// TwinCAT 3 PLC project PlcIotMqttSampleAwsIotShadow
// ProgramVersion: 3.1.4022.7
// libraries:
//   Tc2_Standard, * (Beckhoff Automation GmbH)
//   Tc2_System, * (Beckhoff Automation GmbH)
//   Tc2_Utilities, * (Beckhoff Automation GmbH)
//   Tc3_IotBase, * (Beckhoff Automation GmbH)
//   Tc3_JsonXml, * (Beckhoff Automation GmbH)
//   Tc3_Module, * (Beckhoff Automation GmbH)
// project tree:
//   / PlcTask.TcTTO
//   POUs/ MAIN.TcPOU, PrgMqttCom.TcPOU
// real-time tasks:
//   TASK PlcTask: cycle T#10ms, priority 20, ADS port 350

CONFIGURATION PlcIotMqttSampleAwsIotShadow
    RESOURCE PLC ON TwinCAT3
        TASK PlcTask(INTERVAL := T#10ms, PRIORITY := 20);
        PROGRAM MAIN WITH PlcTask : MAIN;
    END_RESOURCE
END_CONFIGURATION

// ---- POUs/MAIN.TcPOU
PROGRAM MAIN
VAR
	m : INT;
END_VAR

m := m + 1;
PrgMqttCom();

END_PROGRAM

// ---- POUs/PrgMqttCom.TcPOU
PROGRAM PrgMqttCom
VAR
	fbMqttClient 					: FB_IotMqttClient;
	bSetParameter 					: BOOL := TRUE;
	bConnect 						: BOOL := TRUE;
	hrErrorOccurred 				: HRESULT;
	
	(* AWS IoT Shadow  *)
	sTopicShadowUpdate	 			: STRING(255) := '$$aws/things/SvenG-NB05/shadow/update';
	sTopicShadowDocument			: STRING(255) := '$$aws/things/SvenG-NB05/shadow/update/documents';
	sPayloadShadowUpdate			: STRING(1000);
	{attribute 'TcEncoding':='UTF-8'}
	sPayloadShadowDocumentRcv		: STRING(1000);
	bShadowUpdate					: BOOL;
	bShadowDocumentSubscribed		: BOOL;
	
	(* received message and queue handling *)	
	fbMessageQueue 					: FB_IotMqttMessageQueue;
	fbMessage 						: FB_IotMqttMessage;

	(* JSON *)
	fbJson      					: FB_JsonSaxWriter;

END_VAR

IF bSetParameter THEN
	bSetParameter := FALSE;
	
	(* TLS settings for AWS IoT connection *)
	fbMqttClient.stTLS.sCA := 'c:\TwinCAT\3.1\Config\Certificates\AWS\AmazonRootCA1.pem';
    fbMqttClient.stTLS.sCert := 'c:\TwinCAT\3.1\Config\Certificates\AWS\6a1ba937cb-certificate.pem.crt';
    fbMqttClient.stTLS.sKeyFile := 'c:\TwinCAT\3.1\Config\Certificates\AWS\6a1ba937cb-private.pem.key';
	
	(* Broker settings für AWS IoT *)
	fbMqttClient.sHostName:= 'a35rjvy201xp77-ats.iot.eu-central-1.amazonaws.com';
	fbMqttClient.nHostPort:= 8883;
	fbMqttClient.sClientId:= 'SvenG-NB05'; 

	fbMqttClient.ipMessageQueue := fbMessageQueue;
END_IF

fbMqttClient.Execute(bConnect);

IF fbMqttClient.bError THEN
	// add your error logging here
	hrErrorOccurred := fbMqttClient.hrErrorCode;
END_IF
IF fbMessageQueue.nQueuedMessages > 0 THEN
	IF fbMessageQueue.Dequeue(fbMessage:=fbMessage) THEN
		fbMessage.GetTopic(pTopic:=ADR(sTopicShadowDocument), nTopicSize:=SIZEOF(sTopicShadowDocument) );
		fbMessage.GetPayload(pPayload:=ADR(sPayloadShadowDocumentRcv), nPayloadSize:=SIZEOF(sPayloadShadowDocumentRcv), bSetNullTermination:=FALSE);
	END_IF
END_IF

IF fbMqttClient.bConnected THEN
	IF NOT bShadowDocumentSubscribed THEN
		bShadowDocumentSubscribed := fbMqttClient.Subscribe(sTopic:=sTopicShadowDocument, eQoS:=TcIotMqttQos.AtMostOnceDelivery);
		IF fbMqttClient.bError THEN
			// add your error logging here
			hrErrorOccurred := fbMqttClient.hrErrorCode;
		END_IF
	END_IF

	IF bShadowUpdate THEN // update shadow on demand
		bShadowUpdate := FALSE;
		
		// JSON format according to https://docs.aws.amazon.com/iot/latest/developerguide/device-shadow-mqtt.html
		fbJson.StartObject();
		fbJson.AddKey('state');
		fbJson.StartObject();
		fbJson.AddKey('reported');
		fbJson.StartObject();		
		fbJson.AddKey('Vendor');
		fbJson.AddString('Beckhoff Automation');
		fbJson.AddKey('CpuTemperature');
		fbJson.AddDint(42);
		fbJson.AddKey('Operating System');
		fbJson.AddString('FreeBSD');
		fbJson.EndObject();
		fbJson.EndObject();
		fbJson.EndObject();
		sPayloadShadowUpdate := fbJson.GetDocument();
		fbJson.ResetDocument();
	
		fbMqttClient.Publish(	sTopic:= sTopicShadowUpdate, 
								pPayload:= ADR(sPayloadShadowUpdate), nPayloadSize:= LEN2(ADR(sPayloadShadowUpdate)), 
								eQoS:= TcIotMqttQos.AtMostOnceDelivery, bRetain:= FALSE, bQueue:= FALSE );
								
		IF fbMqttClient.bError THEN
				// add your error logging here			
				hrErrorOccurred := fbMqttClient.hrErrorCode;
		END_IF
	END_IF

END_IF

END_PROGRAM
